DATA_BLOCK "dbControl of compressor conection network P2"   // DB53
AUTHOR : rtecmer
VERSION : 0.1
// stored: AutoNumber true, DBAccessibleFromOPCUA true, InstanceOfName Sterowanie dołączeniem na sieć, InstanceOfType FB
"Sterowanie dołączeniem na sieć"
BEGIN
END_DATA_BLOCK

DATA_BLOCK "dbControl of compressor conection network"   // DB47
AUTHOR : rtecmer
VERSION : 0.1
// stored: AutoNumber true, DBAccessibleFromOPCUA true, InstanceOfName Sterowanie dołączeniem na sieć, InstanceOfType FB
"Sterowanie dołączeniem na sieć"
BEGIN
END_DATA_BLOCK

DATA_BLOCK "dbControl of conection network_P1"   // DB54
AUTHOR : rtecmer
VERSION : 0.1
// stored: AutoNumber true, DBAccessibleFromOPCUA true, InstanceOfName Sterowanie dołączeniem na sieć, InstanceOfType FB
"Sterowanie dołączeniem na sieć"
BEGIN
END_DATA_BLOCK

DATA_BLOCK "dbControl of conection network_P3"   // DB55
AUTHOR : rtecmer
VERSION : 0.1
// stored: AutoNumber true, DBAccessibleFromOPCUA true, InstanceOfName Sterowanie dołączeniem na sieć, InstanceOfType FB
"Sterowanie dołączeniem na sieć"
BEGIN
END_DATA_BLOCK

DATA_BLOCK "dbControl of connection Inverters P1"   // DB42
AUTHOR : rtecmer
VERSION : 0.1
// stored: AutoNumber true, DBAccessibleFromOPCUA true, InstanceOfName Sterowanie dołączeniem falownika, InstanceOfType FB
"Sterowanie dołączeniem falownika"
BEGIN
END_DATA_BLOCK

DATA_BLOCK "dbControl of connection Inverters P1_1"   // DB92
AUTHOR : rtecmer
VERSION : 0.1
// stored: AutoNumber true, DBAccessibleFromOPCUA true, InstanceOfName Sterowanie dołączeniem falownika, InstanceOfType FB
"Sterowanie dołączeniem falownika"
BEGIN
END_DATA_BLOCK

DATA_BLOCK "dbControl press oxygen"   // DB64
AUTHOR : rtecmer
VERSION : 0.1
// stored: AutoNumber true, DBAccessibleFromOPCUA true, InstanceOfName Kontrola przekroczenia barMax, InstanceOfType FB
"Kontrola przekroczenia barMax"
BEGIN
END_DATA_BLOCK

DATA_BLOCK "dbControl without inverter"   // DB76
AUTHOR : rtecmer
VERSION : 0.1
// stored: AutoNumber true, DBAccessibleFromOPCUA true, InstanceOfName Sterowania bez falownika, InstanceOfType FB
"Sterowania bez falownika"
BEGIN
END_DATA_BLOCK

DATA_BLOCK "dbControll modors leading and extras"   // DB46
AUTHOR : rtecmer
VERSION : 0.1
// stored: AutoNumber true, DBAccessibleFromOPCUA true, InstanceOfName Ustawienie pomp wiodącej i dodatkowych, InstanceOfType FB
"Ustawienie pomp wiodącej i dodatkowych"
BEGIN
END_DATA_BLOCK

DATA_BLOCK "dbSetup Write Parameters_KDN"   // DB62
AUTHOR : rtecmer
VERSION : 0.1
// stored: AutoNumber true, DBAccessibleFromOPCUA true, InstanceOfName Inicjacja wartości startowych, InstanceOfType FB
"Inicjacja wartości startowych"
BEGIN
END_DATA_BLOCK

DATA_BLOCK "dbSterowanie dołaczaniem dodatkocych_FB1"   // DB3
AUTHOR : RTecmer
FAMILY : Ster
VERSION : 0.1
// stored: AutoNumber true, DBAccessibleFromOPCUA true, InstanceOfName Sterowanie pompami dodatkowymi, InstanceOfType FB
"Sterowanie pompami dodatkowymi"
BEGIN
END_DATA_BLOCK

DATA_BLOCK "dbSterowanie dołączeniem falownika_P4"   // DB33
AUTHOR : rtecmer
VERSION : 0.1
// stored: AutoNumber true, DBAccessibleFromOPCUA true, InstanceOfName Sterowanie dołączeniem falownika, InstanceOfType FB
"Sterowanie dołączeniem falownika"
BEGIN
END_DATA_BLOCK

DATA_BLOCK "dbSterowanie dołączeniem na sieć_P4"   // DB56
AUTHOR : rtecmer
VERSION : 0.1
// stored: AutoNumber true, DBAccessibleFromOPCUA true, InstanceOfName Sterowanie dołączeniem na sieć, InstanceOfType FB
"Sterowanie dołączeniem na sieć"
BEGIN
END_DATA_BLOCK

DATA_BLOCK "dbValueHz_in_Alarm_Pressure_DB"   // DB70
AUTHOR : rtecmer
VERSION : 0.1
// stored: AutoNumber true, DBAccessibleFromOPCUA true, InstanceOfName Kontrola Hz w trybie awayjnym od barMax, InstanceOfType FB
"Kontrola Hz w trybie awayjnym od barMax"
BEGIN
END_DATA_BLOCK

DATA_BLOCK "dbWatchDog HMI"   // DB60
AUTHOR : rtecmer
VERSION : 0.1
// stored: AutoNumber true, DBAccessibleFromOPCUA true, InstanceOfName WatchDog HMI, InstanceOfType FB
"WatchDog HMI"
BEGIN
END_DATA_BLOCK

DATA_BLOCK "dbWatchDog PLC - WinCC"   // DB61
AUTHOR : rtecmer
VERSION : 0.1
// stored: AutoNumber true, DBAccessibleFromOPCUA true, InstanceOfName WatchDog PLC - WinCC, InstanceOfType FB
"WatchDog PLC - WinCC"
BEGIN
END_DATA_BLOCK

DATA_BLOCK "dbcalculation_of_the_increment"   // DB18
AUTHOR : RTecmer
FAMILY : PID
VERSION : 0.1
// stored: AutoNumber true, DBAccessibleFromOPCUA true, InstanceOfName Kontrola przyrostu ciśnieniea, InstanceOfType FB
"Kontrola przyrostu ciśnieniea"
BEGIN
END_DATA_BLOCK

DATA_BLOCK "filtr _kalmana_2_DB_1"   // DB128
VERSION : 0.1
// stored: AutoNumber true, DBAccessibleFromOPCUA true, InstanceOfName filtr _kalmana_2, InstanceOfType FB
"filtr _kalmana_2"
BEGIN
END_DATA_BLOCK

DATA_BLOCK "operating_mode_select_aut-man_DB"   // DB119
AUTHOR : rtecmer
VERSION : 0.1
// stored: AutoNumber true, DBAccessibleFromOPCUA true, InstanceOfName operating_mode_select_aut-man, InstanceOfType FB
"operating_mode_select_aut-man"
BEGIN
END_DATA_BLOCK

DATA_BLOCK "IEC_Timer_AlarmMagistrala_Niskie_DB"   // DB132
{ S7_Optimized_Access := 'TRUE' }
// stored: AutoNumber true, DBAccessibleFromOPCUA true, InstanceOfName IEC_TIMER, OfSystemLibElement IEC_TIMER, OfSystemLibVersion 1.0
"IEC_TIMER"
   // VAR
   //    PT : Time;
   //    ET { ExternalWritable := 'False'} : Time;
   //    IN : Bool;
   //    Q { ExternalWritable := 'False'} : Bool;
   // END_VAR
BEGIN
END_DATA_BLOCK

DATA_BLOCK "IEC_Timer_resetAlarmMagistrala_Niskie_DB"   // DB137
{ S7_Optimized_Access := 'TRUE' }
// stored: AutoNumber true, DBAccessibleFromOPCUA true, InstanceOfName IEC_TIMER, OfSystemLibElement IEC_TIMER, OfSystemLibVersion 1.0
"IEC_TIMER"
   // VAR
   //    PT : Time;
   //    ET { ExternalWritable := 'False'} : Time;
   //    IN : Bool;
   //    Q { ExternalWritable := 'False'} : Bool;
   // END_VAR
BEGIN
END_DATA_BLOCK

DATA_BLOCK "EX012_IDB8_ErrorHandling"   // DB104
VERSION : 0.1
// stored: AutoNumber false, DBAccessibleFromOPCUA true, InstanceOfName EX012_ErrorHandling, InstanceOfType FB
"EX012_ErrorHandling"
   // VAR_INPUT
   //    LED : Int;
   //    CounterError : USInt;
   // END_VAR
   // VAR_OUTPUT
   //    RedLED : Bool;
   // END_VAR
   // VAR
   //    tempCounterDiagStatus : USInt;
   //    tempCounterError : USInt;
   // END_VAR
BEGIN
END_DATA_BLOCK

DATA_BLOCK "FB220_TimeSyn_PLC_To_HMI_DB_1"   // DB78
VERSION : 0.1
// stored: AutoNumber true, DBAccessibleFromOPCUA true, InstanceOfName FB220_TimeSyn_PLC_To_HMI, InstanceOfType FB
"FB220_TimeSyn_PLC_To_HMI"
BEGIN
END_DATA_BLOCK

DATA_BLOCK "HourWork_DB_P1"   // DB5
AUTHOR : RTecmer
FAMILY : XMHour
VERSION : 0.1
// stored: AutoNumber true, DBAccessibleFromOPCUA true, InstanceOfName godzinyPracy, InstanceOfType FB
"godzinyPracy"
BEGIN
END_DATA_BLOCK

DATA_BLOCK "HourWork_P4_DB"   // DB69
AUTHOR : RTecmer
FAMILY : XMHour
VERSION : 0.1
// stored: AutoNumber true, DBAccessibleFromOPCUA true, InstanceOfName godzinyPracy, InstanceOfType FB
"godzinyPracy"
BEGIN
END_DATA_BLOCK

DATA_BLOCK "HourWork__P2_DB"   // DB14
AUTHOR : RTecmer
FAMILY : XMHour
VERSION : 0.1
// stored: AutoNumber true, DBAccessibleFromOPCUA true, InstanceOfName godzinyPracy, InstanceOfType FB
"godzinyPracy"
BEGIN
END_DATA_BLOCK

DATA_BLOCK "HourWork__P3_DB"   // DB15
AUTHOR : RTecmer
FAMILY : XMHour
VERSION : 0.1
// stored: AutoNumber true, DBAccessibleFromOPCUA true, InstanceOfName godzinyPracy, InstanceOfType FB
"godzinyPracy"
BEGIN
END_DATA_BLOCK

DATA_BLOCK "VLV02_Z11_DB"   // DB24
AUTHOR : RTecmer
VERSION : 0.2
// stored: AutoNumber true, DBAccessibleFromOPCUA true, InstanceOfName VLV02, InstanceOfType FB
"VLV02"
BEGIN
END_DATA_BLOCK

DATA_BLOCK "VLV02_Z12_DB"   // DB80
AUTHOR : RTecmer
VERSION : 0.2
// stored: AutoNumber true, DBAccessibleFromOPCUA true, InstanceOfName VLV02, InstanceOfType FB
"VLV02"
BEGIN
END_DATA_BLOCK

DATA_BLOCK "dbModbus_falownik_konwersja"   // DB7
AUTHOR : rtecmer
VERSION : 0.1
// stored: AutoNumber true, DBAccessibleFromOPCUA true, InstanceOfName Konwertowanie parametrów z falownika ModbusRTU, InstanceOfType FB
"Konwertowanie parametrów z falownika ModbusRTU"
BEGIN
END_DATA_BLOCK
